// TIA Portal V16 export
// export: Created 2022-06-06T16:06:40.0293647Z, ExportSetting WithDefaults, DisplayName Totally Integrated Automation Portal, DisplayVersion V16 Update 3, DisplayName TIA Portal Version Control Interface, DisplayVersion V16 Update 2, DisplayName TIA Portal Openness, DisplayVersion V16 Update 3, DisplayName STEP 7 Professional, DisplayVersion V16 Update 3, DisplayName STEP 7 Safety, DisplayVersion V16, DisplayName WinCC Professional, DisplayVersion V16 Update 3
VAR_GLOBAL   // PLC tag table "PAL_FC11011_Test"
   V001_FBK_ENG AT %M100.0 : Bool;   // V001 Energised position limit switch
   V001_FBK_DENG AT %M100.1 : Bool;   // V001 Deenergised position limit switch
   V001_FAULT AT %M100.2 : Bool;   // V001 External fault signal
   V001_OPERATE AT %M101.0 : Bool;   // V001 Energise (operate) signal
   V001_ESTOP AT %M100.3 : Bool;   // V001 Safety signal
   V001_TRIP AT %M100.4 : Bool;   // V001 Trip (interlock) signal
   V001_ILOCK AT %M100.5 : Bool;   // V001 Interlock signal
   V001_PERM AT %M100.6 : Bool;   // V001 Permissive (interlock) signal
   OpTimeRem AT %MD110 : Real;   // Operating timer last non-zero value
END_VAR
